FUNCTION_BLOCK UnitTestSuite IMPLEMENTS ITestSuite
VAR_INPUT
END_VAR
VAR_OUTPUT
END_VAR
VAR
END_VAR

METHOD FB_init : BOOL
VAR_INPUT
	bInitRetains : BOOL; // if TRUE, the retain variables are initialized (warm start / cold start)
	bInCopyCode : BOOL;  // if TRUE, the instance afterwards gets moved into the copy code (online change)
    runner: IRunner;
END_VAR
IF runner <> 0 THEN
    runner.registerTestSuite(THIS^);
END_IF
END_METHOD

PROPERTY numberOfTests : UINT
GET
END_GET
END_PROPERTY

{warning 'add method implementation'}
METHOD runAllTests
END_METHOD

END_FUNCTION_BLOCK

(* stored: Version 1.1.0.1, ProductVersion 3.1.4022.12
   POU UnitTestSuite: Id {fe97e91c-7ea9-4c83-a6e3-45e067042918}, SpecialFunc None
   Method FB_init: Id {6ad6c7a2-2aa4-4197-9227-87f1926f6871}
   Property numberOfTests: Id {8abaee9b-1eb4-4cf9-a836-6101c4e20522}
   Get Get: Id {fd155758-ca70-448f-a471-32b64a788719}
   Method runAllTests: Id {88ad9ea3-be1c-411e-8994-768e609c8491} *)
